FUNCTION FUN_GTAC_GetNodeFromName : String
VAR_INPUT
	InputString:STRING;
	
END_VAR
VAR
	SpaceLoc :INT;
	PeriodLoc:INT;
END_VAR


(*Find the '.' location in the input string *)
PeriodLoc := find(InputString,'.');
SpaceLoc := find(InputString,' ');

(*Using the above location, cut the name out of the input string, and return that as our string*)
IF (SpaceLoc - PeriodLoc) = 5 THEN
	FUN_GTAC_GetNodeFromName:= mid(InputString,4,PeriodLoc+1);
ELSE
	FUN_GTAC_GetNodeFromName:= mid(InputString,3,PeriodLoc+1);
END_IF

END_FUNCTION

(* stored: Version 1.1.0.1, ProductVersion 3.1.4024.9
   POU FUN_GTAC_GetNodeFromName: Id {f20c2dbe-2754-45ae-8e87-1c06add81fcb}, SpecialFunc None *)
